# EPICS autosave request: asiTpxApp/Db/asiTpx_settings.req
file "ADBase_settings.req", P=$(P), R=$(R)
$(P)$(R)TDC1Enable
$(P)$(R)TDC1Edge
$(P)$(R)TDC1Output
$(P)$(R)TDC2Enable
$(P)$(R)TDC2Edge
$(P)$(R)TDC2Output
$(P)$(R)TriggerPolarity
$(P)$(R)RawEnable
$(P)$(R)RawFilePath
$(P)$(R)RawFileTemplate
$(P)$(R)ImageEnable
$(P)$(R)ImageFilePath
$(P)$(R)ImageFileTemplate
$(P)$(R)PixelMode
$(P)$(R)DataSource
$(P)$(R)PreviewPeriod
